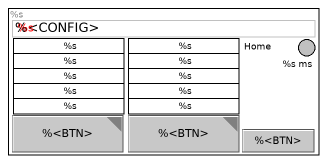
[picture p238: ZLIB_VALVE_5_SENSORS (HMI screen)]
rectangle at (0,0)-(311,147): text "%s"; shows $Object$.BitName
rectangle at (5,30)-(116,46): text "%s"; shows $Object$.SAInitPosName; invisible if $Object$.NoOfInitSensors<1; alarm colour if $Object$.AInitPosition; dynamic style TRUE
rectangle at (5,45)-(116,61): text "%s"; shows $Object$.SBInitPosName; invisible if $Object$.NoOfInitSensors<2; alarm colour if $Object$.BInitPosition; dynamic style TRUE
rectangle at (120,30)-(231,46): text "%s"; shows $Object$.SAWorkPosName; invisible if $Object$.NoOfWorkSensors<1; alarm colour if $Object$.AWorkPosition; dynamic style TRUE
rectangle at (120,45)-(231,61): text "%s"; shows $Object$.SBWorkPosName; invisible if $Object$.NoOfWorkSensors<2; alarm colour if $Object$.BWorkPosition; dynamic style TRUE
ellipse at (290,31)-(307,48): alarm colour if $Object$.HomePosition; dynamic style TRUE
rounded rectangle at (234,32)-(280,45): text "Home"; shows $Object$.State
rectangle at (235,48)-(306,64): text "%s ms"; shows $Object$.ProcessTime
rectangle at (5,60)-(116,76): text "%s"; shows $Object$.SCInitPosName; invisible if $Object$.NoOfInitSensors<3; alarm colour if $Object$.CInitPosition; dynamic style TRUE
rectangle at (120,60)-(231,76): text "%s"; shows $Object$.SCWorkPosName; invisible if $Object$.NoOfWorkSensors<3; alarm colour if $Object$.CWorkPosition; dynamic style TRUE
rectangle at (5,75)-(116,91): text "%s"; shows $Object$.SDInitPosName; invisible if $Object$.NoOfInitSensors<4; alarm colour if $Object$.DInitPosition; dynamic style TRUE
rectangle at (120,75)-(231,91): text "%s"; shows $Object$.SDWorkPosName; invisible if $Object$.NoOfWorkSensors<4; alarm colour if $Object$.DWorkPosition; dynamic style TRUE
rectangle at (5,90)-(116,106): text "%s"; shows $Object$.SEInitPosName; invisible if $Object$.NoOfInitSensors<5; alarm colour if $Object$.EInitPosition; dynamic style TRUE
rectangle at (120,90)-(231,106): text "%s"; shows $Object$.SEWorkPosName; invisible if $Object$.NoOfWorkSensors<5; alarm colour if $Object$.EWorkPosition; dynamic style TRUE
button at (234,121)-(306,144): text "%<BTN>"; shows $Object$.BtnReset.Text; invisible if NOT $Object$.BtnReset.Visible; taps $Object$.BtnReset.Pressed; dynamic style $Object$.BtnReset.TextColor, $Object$.BtnReset.BackgroundColor, $Object$.BtnReset.BackgroundColor, NOT $Object$.BtnReset.Enable
button at (120,107)-(231,144): text "%<BTN>"; shows $Object$.BtnMoveWork.Text; invisible if NOT $Object$.BtnMoveWork.Visible; taps $Object$.BtnMoveWork.Pressed; dynamic style $Object$.BtnMoveWork.TextColor, $Object$.BtnMoveWork.BackgroundColor, $Object$.BtnMoveWork.BackgroundColor, NOT $Object$.BtnMoveWork.Enable
button at (4,107)-(115,144): text "%<BTN>"; shows $Object$.BtnMoveInit.Text; invisible if NOT $Object$.BtnMoveInit.Visible; taps $Object$.BtnMoveInit.Pressed; dynamic style $Object$.BtnMoveInit.TextColor, $Object$.BtnMoveInit.BackgroundColor, $Object$.BtnMoveInit.BackgroundColor, NOT $Object$.BtnMoveInit.Enable
rectangle at (5,11)-(306,28): text "%<CONFIG>"; shows $Object$.InstName
rounded rectangle at (4,12)-(307,29): text "%s"; shows $Object$.ErrorString; invisible if NOT $Object$.ErrorPresent
polygon at (99,109)-(113,123): invisible if $Object$.NoOfValveCoils<2; alarm colour if $Object$.CoilB
polygon at (215,109)-(229,123): alarm colour if $Object$.CoilA
*)

(* Visualisation ZLIB_SERVICELINE
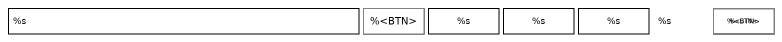
rectangle at (0,0)-(351,26): text "%s"; shows Service.daten[$Object$].Name; editable; dynamic style ST_Service.ColorName[$Object$], $deaktivieren$
embedded screen at (355,0)-(416,26): ZLIB_VISUBUTTON_TOGGELN
rectangle at (495,0)-(566,26): text "%s"; shows Service.daten[$Object$].Warning_Value; editable 0..; dynamic style $deaktivieren$
embedded screen at (705,0)-(766,26): ZLIB_VISUBUTTON
rectangle at (420,0)-(491,26): text "%s"; shows Service.daten[$Object$].Default_Value; editable 0..; dynamic style $deaktivieren$
rectangle at (570,0)-(641,26): text "%s"; shows Service.visu[$Object$].Current_Value; dynamic style Service.visu[$Object$].Current_Value_Color
rectangle at (645,0)-(706,26): text "%s"; shows Service.daten[$Object$].Unit
embedded screen at (705,0)-(766,26): ZLIB_VISUBUTTON_S17
rectangle at (0,0)-(351,26): text "%s"; shows Service.daten[$Object$].Name; invisible if $deaktivieren$; editable; dynamic style ST_Service.ColorName[$Object$], $deaktivieren$
rectangle at (495,0)-(566,26): text "%s"; shows Service.daten[$Object$].Warning_Value; invisible if $deaktivieren$; editable 0..; dynamic style $deaktivieren$
rectangle at (420,0)-(491,26): text "%s"; shows Service.daten[$Object$].Default_Value; invisible if $deaktivieren$; editable 0..; dynamic style $deaktivieren$
*)

(* Visualisation ZLIB_SERVICELIST
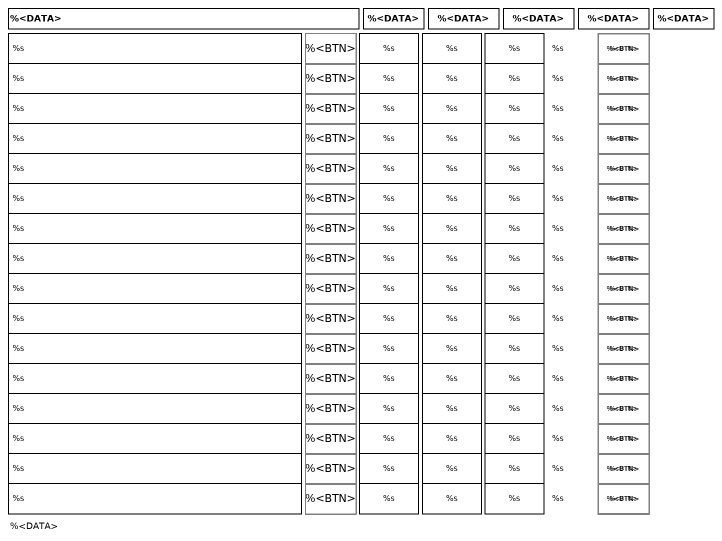
embedded screen at (0,25)-(641,56): ZLIB_SERVICELINE
embedded screen at (0,55)-(641,86): ZLIB_SERVICELINE
rectangle at (0,0)-(351,21): text "%<DATA>"; shows 'Bezeichung der Wartung'
rectangle at (355,0)-(416,21): text "%<DATA>"; shows 'Art'
rectangle at (420,0)-(491,21): text "%<DATA>"; shows 'Vorgabe'
rectangle at (495,0)-(566,21): text "%<DATA>"; shows 'Warngrenze'
rectangle at (570,0)-(641,21): text "%<DATA>"; shows 'Aktuell'
rectangle at (645,0)-(706,21): text "%<DATA>"; shows 'Einheit'
embedded screen at (0,85)-(641,116): ZLIB_SERVICELINE
embedded screen at (0,115)-(641,146): ZLIB_SERVICELINE
embedded screen at (0,145)-(641,176): ZLIB_SERVICELINE
embedded screen at (0,175)-(641,206): ZLIB_SERVICELINE
embedded screen at (0,205)-(641,236): ZLIB_SERVICELINE
embedded screen at (0,235)-(641,266): ZLIB_SERVICELINE
embedded screen at (0,265)-(641,296): ZLIB_SERVICELINE
embedded screen at (0,295)-(641,326): ZLIB_SERVICELINE
embedded screen at (0,325)-(641,356): ZLIB_SERVICELINE
embedded screen at (0,355)-(641,386): ZLIB_SERVICELINE
embedded screen at (0,385)-(641,416): ZLIB_SERVICELINE
embedded screen at (0,415)-(641,446): ZLIB_SERVICELINE
embedded screen at (0,445)-(641,476): ZLIB_SERVICELINE
embedded screen at (0,475)-(641,506): ZLIB_SERVICELINE
rectangle at (0,505)-(766,531): text "%<DATA>"; shows 'Info'
*)

(* Visualisation ZLIB_VISUBUTTON_TOGGELN
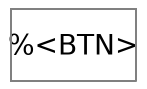
rectangle at (0,0)-(126,73): text "%<BTN>"; shows $Object$.Text; invisible if NOT $Object$.Visible; alarm colour if NOT $Object$.Enable; taps $Object$.Pressed; dynamic style $Object$.TextColor, $Object$.BackgroundColor, $Object$.BackgroundColor, NOT $Object$.Enable
polyline at (125,1)-(125,72): invisible if NOT $Object$.Visible; alarm colour if $Object$.Pressed
polyline at (1,72)-(125,72): invisible if NOT $Object$.Visible; alarm colour if $Object$.Pressed
polyline at (1,1)-(125,1): invisible if NOT $Object$.Visible; alarm colour if NOT $Object$.Pressed
polyline at (1,1)-(1,72): invisible if NOT $Object$.Visible; alarm colour if NOT $Object$.Pressed
polyline at (0,73)-(126,73): invisible if NOT $Object$.Visible; alarm colour if $Object$.Pressed
polyline at (126,0)-(126,73): invisible if NOT $Object$.Visible; alarm colour if $Object$.Pressed
polyline at (0,0)-(126,0): invisible if NOT $Object$.Visible; alarm colour if NOT $Object$.Pressed
polyline at (0,0)-(0,73): invisible if NOT $Object$.Visible; alarm colour if NOT $Object$.Pressed
*)

(* Visualisation INFO_TREE
rounded rectangle at (0,0)-(161,21): text "%<TREE>"; shows $Objekt$.Text; invisible if $Objekt$.unsichtbar; taps $Objekt$.tasten; opens $Objekt$.Zoom; dynamic style $Objekt$.TextFarbe, $Objekt$.deaktivieren
*)

(* Visualisation VISUBUTTON_TREE
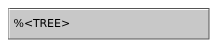
button at (0,0)-(201,31): text "%<TREE>"; shows $Objekt$.Text; invisible if $Objekt$.unsichtbar; taps $Objekt$.tasten; opens $Objekt$.Zoom; dynamic style $Objekt$.TextFarbe, $Objekt$.innenFarbe, $Objekt$.innenFarbe, $Objekt$.deaktivieren
*)

(* Visualisation ZLIB_SFC_STATE
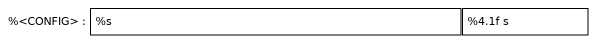
rectangle at (0,0)-(231,27): text "%<CONFIG> :"; shows $SFC$.SFCCurrentPOU
rectangle at (230,0)-(601,27): text "%s"; shows $SFC$.SFCCurrentStep
rectangle at (602,0)-(728,27): text "%4.1f s"; shows $SFC$.SFCTime / 1000.0
*)

(* Visualisation ZLIB_VISUBUTTON
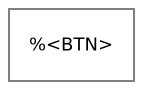
rectangle at (0,0)-(126,73): text "%<BTN>"; shows $Object$.Text; invisible if NOT $Object$.Visible; alarm colour if NOT $Object$.Enable; taps $Object$.Pressed; dynamic style $Object$.TextColor, $Object$.BackgroundColor, $Object$.BackgroundColor, NOT $Object$.Enable
polyline at (125,1)-(125,72): invisible if NOT $Object$.Visible; alarm colour if $Object$.Pressed
polyline at (1,72)-(125,72): invisible if NOT $Object$.Visible; alarm colour if $Object$.Pressed
polyline at (1,1)-(125,1): invisible if NOT $Object$.Visible; alarm colour if NOT $Object$.Pressed
polyline at (1,1)-(1,72): invisible if NOT $Object$.Visible; alarm colour if NOT $Object$.Pressed
polyline at (0,73)-(126,73): invisible if NOT $Object$.Visible; alarm colour if $Object$.Pressed
polyline at (126,0)-(126,73): invisible if NOT $Object$.Visible; alarm colour if $Object$.Pressed
polyline at (0,0)-(126,0): invisible if NOT $Object$.Visible; alarm colour if NOT $Object$.Pressed
polyline at (0,0)-(0,73): invisible if NOT $Object$.Visible; alarm colour if NOT $Object$.Pressed
*)

(* Visualisation ZLIB_VISUBUTTON_ARROW_DOWN
polygon at (2,2)-(102,82): text "%s"; shows $Object$.Text; invisible if NOT $Object$.Visible; alarm colour if NOT $Object$.Enable; taps $Object$.Pressed; dynamic style $Object$.BackgroundColor, $Object$.BackgroundColor, NOT $Object$.Enable
*)

(* Visualisation ZLIB_VISUBUTTON_ARROW_UP
polygon at (2,2)-(102,82): text "%s"; shows $Object$.Text; invisible if NOT $Object$.Visible; alarm colour if NOT $Object$.Enable; taps $Object$.Pressed; dynamic style $Object$.BackgroundColor, $Object$.BackgroundColor, NOT $Object$.Enable
*)

(* Visualisation ZLIB_VISUBUTTON_MODE_SELECT
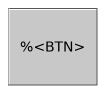
button at (0,0)-(89,77): text "%<BTN>"; shows $Object$.Text; invisible if NOT $Object$.Visible; taps $Object$.Pressed; dynamic style $Object$.TextColor, $Object$.BackgroundColor, $Object$.BackgroundColor, NOT $Object$.Enable
*)

(* Visualisation ZLIB_VISUBUTTON_S17
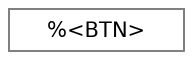
rectangle at (0,0)-(176,43): text "%<BTN>"; shows $Object$.Text; invisible if NOT $Object$.Visible; alarm colour if NOT $Object$.Enable; taps $Object$.Pressed; dynamic style $Object$.TextColor, $Object$.BackgroundColor, $Object$.BackgroundColor, NOT $Object$.Enable
polyline at (175,1)-(175,42): invisible if NOT $Object$.Visible; alarm colour if $Object$.Pressed
polyline at (1,42)-(175,42): invisible if NOT $Object$.Visible; alarm colour if $Object$.Pressed
polyline at (1,1)-(175,1): invisible if NOT $Object$.Visible; alarm colour if NOT $Object$.Pressed
polyline at (1,1)-(1,42): invisible if NOT $Object$.Visible; alarm colour if NOT $Object$.Pressed
polyline at (0,43)-(176,43): invisible if NOT $Object$.Visible; alarm colour if $Object$.Pressed
polyline at (176,0)-(176,43): invisible if NOT $Object$.Visible; alarm colour if $Object$.Pressed
polyline at (0,0)-(176,0): invisible if NOT $Object$.Visible; alarm colour if NOT $Object$.Pressed
polyline at (0,0)-(0,43): invisible if NOT $Object$.Visible; alarm colour if NOT $Object$.Pressed
*)

(* Visualisation ZLIB_VISUBUTTON_S18
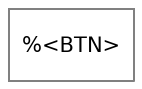
rectangle at (0,0)-(126,73): text "%<BTN>"; shows $Object$.Text; invisible if NOT $Object$.Visible; alarm colour if NOT $Object$.Enable; taps $Object$.Pressed; dynamic style $Object$.TextColor, $Object$.BackgroundColor, $Object$.BackgroundColor, NOT $Object$.Enable
polyline at (125,1)-(125,72): invisible if NOT $Object$.Visible; alarm colour if $Object$.Pressed
polyline at (1,72)-(125,72): invisible if NOT $Object$.Visible; alarm colour if $Object$.Pressed
polyline at (1,1)-(125,1): invisible if NOT $Object$.Visible; alarm colour if NOT $Object$.Pressed
polyline at (1,1)-(1,72): invisible if NOT $Object$.Visible; alarm colour if NOT $Object$.Pressed
polyline at (0,73)-(126,73): invisible if NOT $Object$.Visible; alarm colour if $Object$.Pressed
polyline at (126,0)-(126,73): invisible if NOT $Object$.Visible; alarm colour if $Object$.Pressed
polyline at (0,0)-(126,0): invisible if NOT $Object$.Visible; alarm colour if NOT $Object$.Pressed
polyline at (0,0)-(0,73): invisible if NOT $Object$.Visible; alarm colour if NOT $Object$.Pressed
*)

(* Visualisation ZLIB_VISUBUTTON_S24
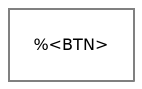
rectangle at (0,0)-(126,73): text "%<BTN>"; shows $Object$.Text; invisible if NOT $Object$.Visible; alarm colour if NOT $Object$.Enable; taps $Object$.Pressed; dynamic style $Object$.TextColor, $Object$.BackgroundColor, $Object$.BackgroundColor, NOT $Object$.Enable
polyline at (125,1)-(125,72): invisible if NOT $Object$.Visible; alarm colour if $Object$.Pressed
polyline at (1,72)-(125,72): invisible if NOT $Object$.Visible; alarm colour if $Object$.Pressed
polyline at (1,1)-(125,1): invisible if NOT $Object$.Visible; alarm colour if NOT $Object$.Pressed
polyline at (1,1)-(1,72): invisible if NOT $Object$.Visible; alarm colour if NOT $Object$.Pressed
polyline at (0,73)-(126,73): invisible if NOT $Object$.Visible; alarm colour if $Object$.Pressed
polyline at (126,0)-(126,73): invisible if NOT $Object$.Visible; alarm colour if $Object$.Pressed
polyline at (0,0)-(126,0): invisible if NOT $Object$.Visible; alarm colour if NOT $Object$.Pressed
polyline at (0,0)-(0,73): invisible if NOT $Object$.Visible; alarm colour if NOT $Object$.Pressed
*)

(* Visualisation ZLIB_VISUBUTTON_S24_S
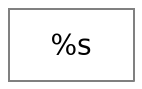
rectangle at (0,0)-(126,73): text "%s"; shows $Object$.Text; invisible if NOT $Object$.Visible; alarm colour if NOT $Object$.Enable; taps $Object$.Pressed; dynamic style $Object$.TextColor, $Object$.BackgroundColor, $Object$.BackgroundColor, NOT $Object$.Enable
polyline at (125,1)-(125,72): invisible if NOT $Object$.Visible; alarm colour if $Object$.Pressed
polyline at (1,72)-(125,72): invisible if NOT $Object$.Visible; alarm colour if $Object$.Pressed
polyline at (1,1)-(125,1): invisible if NOT $Object$.Visible; alarm colour if NOT $Object$.Pressed
polyline at (1,1)-(1,72): invisible if NOT $Object$.Visible; alarm colour if NOT $Object$.Pressed
polyline at (0,73)-(126,73): invisible if NOT $Object$.Visible; alarm colour if $Object$.Pressed
polyline at (126,0)-(126,73): invisible if NOT $Object$.Visible; alarm colour if $Object$.Pressed
polyline at (0,0)-(126,0): invisible if NOT $Object$.Visible; alarm colour if NOT $Object$.Pressed
polyline at (0,0)-(0,73): invisible if NOT $Object$.Visible; alarm colour if NOT $Object$.Pressed
*)

(* Visualisation ZLIB_VISUBUTTON_S24_S_IO
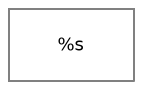
rectangle at (0,0)-(126,73): text "%s"; shows $Object$.Text; invisible if NOT $Object$.Visible; alarm colour if NOT $Object$.Enable; taps $Object$.Pressed; dynamic style $Object$.TextColor, $Object$.BackgroundColor, $Object$.BackgroundColor, NOT $Object$.Enable
polyline at (125,1)-(125,72): invisible if NOT $Object$.Visible; alarm colour if $Object$.Pressed
polyline at (1,72)-(125,72): invisible if NOT $Object$.Visible; alarm colour if $Object$.Pressed
polyline at (1,1)-(125,1): invisible if NOT $Object$.Visible; alarm colour if NOT $Object$.Pressed
polyline at (1,1)-(1,72): invisible if NOT $Object$.Visible; alarm colour if NOT $Object$.Pressed
polyline at (0,73)-(126,73): invisible if NOT $Object$.Visible; alarm colour if $Object$.Pressed
polyline at (126,0)-(126,73): invisible if NOT $Object$.Visible; alarm colour if $Object$.Pressed
polyline at (0,0)-(126,0): invisible if NOT $Object$.Visible; alarm colour if NOT $Object$.Pressed
polyline at (0,0)-(0,73): invisible if NOT $Object$.Visible; alarm colour if NOT $Object$.Pressed
*)

(* Visualisation ZLIB_VISUBUTTON_S36
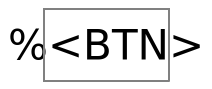
rectangle at (0,0)-(126,73): text "%<BTN>"; shows $Object$.Text; invisible if NOT $Object$.Visible; alarm colour if NOT $Object$.Enable; taps $Object$.Pressed; dynamic style $Object$.TextColor, $Object$.BackgroundColor, $Object$.BackgroundColor, NOT $Object$.Enable
polyline at (125,1)-(125,72): invisible if NOT $Object$.Visible; alarm colour if $Object$.Pressed
polyline at (1,72)-(125,72): invisible if NOT $Object$.Visible; alarm colour if $Object$.Pressed
polyline at (1,1)-(125,1): invisible if NOT $Object$.Visible; alarm colour if NOT $Object$.Pressed
polyline at (1,1)-(1,72): invisible if NOT $Object$.Visible; alarm colour if NOT $Object$.Pressed
polyline at (0,73)-(126,73): invisible if NOT $Object$.Visible; alarm colour if $Object$.Pressed
polyline at (126,0)-(126,73): invisible if NOT $Object$.Visible; alarm colour if $Object$.Pressed
polyline at (0,0)-(126,0): invisible if NOT $Object$.Visible; alarm colour if NOT $Object$.Pressed
polyline at (0,0)-(0,73): invisible if NOT $Object$.Visible; alarm colour if NOT $Object$.Pressed
*)

(* Visualisation ZLIBVISUBUTTON_TEXTINPUT
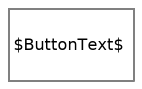
rectangle at (0,0)-(126,73): text "$ButtonText$"; shows $InputVar$; invisible if NOT $Object$.Visible; alarm colour if NOT $Object$.Enable; editable; dynamic style $Object$.TextColor, $Object$.BackgroundColor, $Object$.BackgroundColor, NOT $Object$.Enable
polyline at (125,1)-(125,72): invisible if NOT $Object$.Visible; alarm colour if $Object$.Pressed
polyline at (1,72)-(125,72): invisible if NOT $Object$.Visible; alarm colour if $Object$.Pressed
polyline at (1,1)-(125,1): invisible if NOT $Object$.Visible; alarm colour if NOT $Object$.Pressed
polyline at (1,1)-(1,72): invisible if NOT $Object$.Visible; alarm colour if NOT $Object$.Pressed
polyline at (0,73)-(126,73): invisible if NOT $Object$.Visible; alarm colour if $Object$.Pressed
polyline at (126,0)-(126,73): invisible if NOT $Object$.Visible; alarm colour if $Object$.Pressed
polyline at (0,0)-(126,0): invisible if NOT $Object$.Visible; alarm colour if NOT $Object$.Pressed
polyline at (0,0)-(0,73): invisible if NOT $Object$.Visible; alarm colour if NOT $Object$.Pressed
*)

(* Visualisation ZLIBVISUBUTTON_TEXTVAR
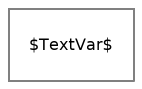
rectangle at (0,0)-(126,73): text "$TextVar$"; shows $TextVar$; invisible if NOT $Object$.Visible; alarm colour if NOT $Object$.Enable; taps $Object$.Pressed; dynamic style $Object$.TextColor, $Object$.BackgroundColor, $Object$.BackgroundColor, NOT $Object$.Enable
polyline at (125,1)-(125,72): invisible if NOT $Object$.Visible; alarm colour if $Object$.Pressed
polyline at (1,72)-(125,72): invisible if NOT $Object$.Visible; alarm colour if $Object$.Pressed
polyline at (1,1)-(125,1): invisible if NOT $Object$.Visible; alarm colour if NOT $Object$.Pressed
polyline at (1,1)-(1,72): invisible if NOT $Object$.Visible; alarm colour if NOT $Object$.Pressed
polyline at (0,73)-(126,73): invisible if NOT $Object$.Visible; alarm colour if $Object$.Pressed
polyline at (126,0)-(126,73): invisible if NOT $Object$.Visible; alarm colour if $Object$.Pressed
polyline at (0,0)-(126,0): invisible if NOT $Object$.Visible; alarm colour if NOT $Object$.Pressed
polyline at (0,0)-(0,73): invisible if NOT $Object$.Visible; alarm colour if NOT $Object$.Pressed
*)

(* Visualisation ZLIBVISUBUTTON_ZOOMTOCALLER
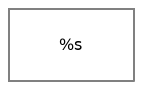
rectangle at (0,0)-(126,73): text "%s"; shows $Object$.Text; invisible if NOT $Object$.Visible; alarm colour if NOT $Object$.Enable; taps $Object$.Pressed; opens ZOOMTOCALLER; dynamic style $Object$.TextColor, $Object$.BackgroundColor, $Object$.BackgroundColor, NOT $Object$.Enable
polyline at (125,1)-(125,72): invisible if NOT $Object$.Visible; alarm colour if $Object$.Pressed
polyline at (1,72)-(125,72): invisible if NOT $Object$.Visible; alarm colour if $Object$.Pressed
polyline at (1,1)-(125,1): invisible if NOT $Object$.Visible; alarm colour if NOT $Object$.Pressed
polyline at (1,1)-(1,72): invisible if NOT $Object$.Visible; alarm colour if NOT $Object$.Pressed
polyline at (0,73)-(126,73): invisible if NOT $Object$.Visible; alarm colour if $Object$.Pressed
polyline at (126,0)-(126,73): invisible if NOT $Object$.Visible; alarm colour if $Object$.Pressed
polyline at (0,0)-(126,0): invisible if NOT $Object$.Visible; alarm colour if NOT $Object$.Pressed
polyline at (0,0)-(0,73): invisible if NOT $Object$.Visible; alarm colour if NOT $Object$.Pressed
*)

(* Visualisation WPC_CONVEYOR_IN
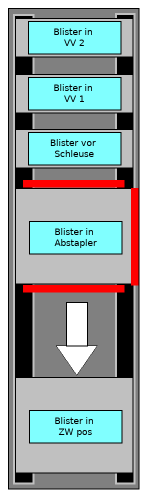
embedded screen at (48,294)-(89,367): SIGNS_ARROWDOWN
rectangle at (7,180)-(125,276): text "%<BASIC>"; shows 'Blister in Abstapler'; alarm colour if NOT ST08_404_B52_2.BitInToCheck; opens Visu.MainMenue.BtnManual_ST08_2.zoom
rectangle at (7,369)-(125,465): text "%<BASIC>"; shows 'Blister in ZW pos'; alarm colour if NOT ST08_406_B54_0.BitInToCheck; opens Visu.MainMenue.BtnManual_ST08_3.zoom
rectangle at (7,121)-(125,160): text "%<BASIC>"; shows 'Blister vor Schleuse'; alarm colour if NOT ST08_402_B51_2.BitInToCheck; opens Visu.MainMenue.BtnManual_ST08_1.zoom
rectangle at (7,66)-(125,105): text "%<BASIC>"; shows 'Blister in VV1'; invisible if NOT .MP.ST08.Trayzufuhr_Verlaengerung; alarm colour if NOT ST08_401_B50_5.BitInToCheck; opens Visu.MainMenue.BtnManual_ST08_1.zoom
rectangle at (7,10)-(125,49): text "%<BASIC>"; shows 'Blister in VV2'; invisible if NOT .MP.ST08.Trayzufuhr_Verlaengerung; alarm colour if NOT ST08_400_B50_0.BitInToCheck; opens Visu.MainMenue.BtnManual_ST08_1.zoom
rectangle at (20,13)-(113,46): text "Blister in / VV 2"; invisible if TRUE
rectangle at (20,69)-(113,102): text "Blister in / VV 1"; invisible if TRUE
rectangle at (20,124)-(113,157): text "Blister vor / Schleuse"; invisible if TRUE
rectangle at (21,213)-(114,246): text "Blister in / Abstapler"; invisible if TRUE
rectangle at (21,402)-(114,435): text "Blister in / ZW pos"; invisible if TRUE
embedded screen at (123,180)-(130,277): DOOR_LOCK; tooltip ST00_229_S1
embedded screen at (15,172)-(116,179): DOOR_LOCK; tooltip ST00_226_S1
embedded screen at (15,277)-(116,284): DOOR_LOCK; tooltip ST00_226_S2
3 more shapes without text or variables
*)

(* Visualisation WPC_CONVEYOR_OUT
embedded screen at (49,4294967295)-(90,72): Signs_ArrowUp
rectangle at (7,61)-(125,100): text "%<BASIC>"; shows 'Stau im Auslauf'; alarm colour if NOT ST08_409_B55_5.BitInToCheck
rectangle at (25,64)-(118,97): text "Stau im / Auslauf"; invisible if TRUE
embedded screen at (7,370)-(129,468): WPC_OUT; shows TD.PartsInBlisterInlet; opens Visu.MainMenue.BtnManual_ST08_3.zoom
embedded screen at (7,183)-(125,284): WPC_OUT_AUFSTAPELN; shows TD.PartsInBlisterInlet; opens Visu.MainMenue.BtnManual_ST08_4.zoom
embedded screen at (7,183)-(14,280): DOOR_LOCK; tooltip ST00_230_S1
embedded screen at (15,176)-(116,183): DOOR_LOCK; tooltip ST00_227_S1
embedded screen at (15,281)-(116,288): DOOR_LOCK; tooltip ST00_227_S2
embedded screen at (0,181)-(7,282): DOOR_LOCK; tooltip ST00_232_S1
3 more shapes without text or variables
*)

(* Visualisation WPC_OUT
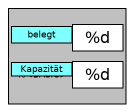
rectangle at (0,0)-(118,96): alarm colour if NOT ST08_406_B54_3.BitInToCheck OR ST08_406_B54_4.ValveSensor
rectangle at (64,16)-(115,43): text "%d"; shows PosIdx-TD.PartsInRoboGripper
rectangle at (2,16)-(64,43): text "%<BASIC>"; shows 'belegt'
rectangle at (64,53)-(115,80): text "%d"; shows TD.PartsInBlisterInlet
rectangle at (2,53)-(64,80): text "%<BASIC>"; shows 'Kapazität'
rectangle at (64,16)-(115,43): shows ST08_CallPRGs.PosIdxHelp; editable 0..TD.PartsInBlisterInlet
rectangle at (3,18)-(64,35): text "belegt"; invisible if TRUE
rectangle at (3,54)-(64,68): text "Kapazität"; invisible if TRUE
rectangle at (64,16)-(115,43): text "%d"; shows PosIdx-TD.PartsInRoboGripper; invisible if $deaktivieren$
*)

(* Visualisation WPC_OUT_AUFSTAPELN
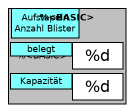
rectangle at (0,0)-(118,96): alarm colour if NOT ST08_407_B55_4.BitInToCheck
rectangle at (2,34)-(64,61): text "%<BASIC>"; shows 'belegt'
rectangle at (64,65)-(115,92): text "%d"; shows .TD.NoOfPalletsPerStack; editable 0..
rectangle at (2,65)-(64,92): text "%<BASIC>"; shows 'Kapazität'
rectangle at (2,34)-(64,48): text "belegt"; invisible if TRUE
rectangle at (2,65)-(64,81): text "Kapazität"; invisible if TRUE
rectangle at (3,0)-(71,30): text "Aufstapeln / Anzahl Blister"; invisible if TRUE
rectangle at (0,3)-(118,31): text "%<BASIC>"; shows 'Aufstapeln Anzahl Blister'
rectangle at (64,34)-(115,61): text "%d"; shows .MP.ST08.NoOfBlisterInStackerOut; editable 0...TD.NoOfPalletsPerStack; dynamic style $deaktivieren$
rectangle at (64,34)-(115,61): text "%d"; shows .MP.ST08.NoOfBlisterInStackerOut; invisible if $deaktivieren$; editable 0...TD.NoOfPalletsPerStack
*)

(* Visualisation ROUNDTABLE
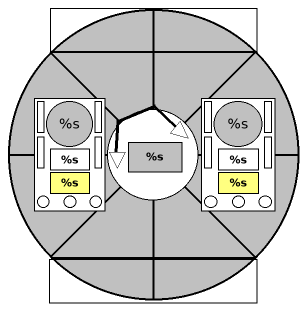
polyline at (147,3)-(147,291): invisible if (ST02_DT_62_B81.ValveSensor OR ST02_DT_62_B91.ValveSensor)
polyline at (2,147)-(292,147): invisible if (ST02_DT_62_B81.ValveSensor OR ST02_DT_62_B91.ValveSensor)
polyline at (44,44)-(249,249): invisible if NOT (ST02_DT_62_B81.ValveSensor OR ST02_DT_62_B91.ValveSensor)
polyline at (44,44)-(249,249): invisible if NOT (ST02_DT_62_B81.ValveSensor OR ST02_DT_62_B91.ValveSensor)
embedded screen at (195,90)-(269,203): RoundTableNest
embedded screen at (28,90)-(99,203): ROUNDTABLENEST
polygon at (103,144)-(119,160): alarm colour if ST02_62_Y6.MoveWork
rounded rectangle at (122,134)-(176,164): text "%s"; shows MachineStates.CycleTimeHelp
polygon at (164,113)-(182,130): alarm colour if ST02_62_Y6.MoveInit
7 more shapes without text or variables
*)

(* Visualisation ROUNDTABLE_1
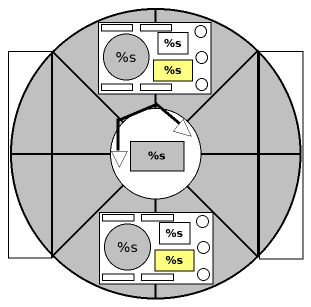
polyline at (147,3)-(147,291): invisible if (ST02_DT_62_B81.ValveSensor OR ST02_DT_62_B91.ValveSensor)
polyline at (2,147)-(292,147): invisible if (ST02_DT_62_B81.ValveSensor OR ST02_DT_62_B91.ValveSensor)
polyline at (44,44)-(249,249): invisible if NOT (ST02_DT_62_B81.ValveSensor OR ST02_DT_62_B91.ValveSensor)
polyline at (44,44)-(249,249): invisible if NOT (ST02_DT_62_B81.ValveSensor OR ST02_DT_62_B91.ValveSensor)
embedded screen at (90,14)-(203,87): RoundTableNest_1
embedded screen at (91,204)-(205,277): ROUNDTABLENEST_1
polygon at (103,144)-(119,160): alarm colour if ST02_62_Y6.MoveWork
rounded rectangle at (122,134)-(176,164): text "%s"; shows MachineStates.CycleTimeHelp
polygon at (165,112)-(183,129): alarm colour if ST02_62_Y6.MoveInit
7 more shapes without text or variables
*)

(* Visualisation ROUNDTABLENEST
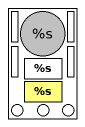
ellipse at (12,3)-(57,48): text "%s"; shows $NestNo$; invisible if NOT MP.ST02.TableData[$NestNo$].ProcessData.Part; alarm colour if MP.ST02.TableData[$NestNo$].ProcessData.Result >11; toggles MP.ST02.TableData[$NestNo$].ProcessData.Part
ellipse at (12,3)-(57,48): text "%s"; shows $NestNo$; invisible if MP.ST02.TableData[$NestNo$].ProcessData.Part; toggles MP.ST02.TableData[$NestNo$].ProcessData.Part
rectangle at (16,73)-(54,94): text "%s"; shows MP.ST02.TableData[$NestNo$].ProcessData.Result; editable
rectangle at (3,38)-(10,69): invisible if NOT MP.ST02.TableData[$NestNo$].ProcessData.Part OR MP.ST02.TableData[$NestNo$].ProcessData.Result >=19; alarm colour if MP.ST02.TableData[$NestNo$].ProcessData.Result >=1
rectangle at (3,3)-(10,34): invisible if NOT MP.ST02.TableData[$NestNo$].ProcessData.Part OR MP.ST02.TableData[$NestNo$].ProcessData.Result >=19; alarm colour if MP.ST02.TableData[$NestNo$].ProcessData.Result >=1
rectangle at (59,38)-(66,69): invisible if NOT MP.ST02.TableData[$NestNo$].ProcessData.Part OR MP.ST02.TableData[$NestNo$].ProcessData.Result >=19; alarm colour if MP.ST02.TableData[$NestNo$].ProcessData.Result >=11
rectangle at (59,3)-(66,34): invisible if NOT MP.ST02.TableData[$NestNo$].ProcessData.Part OR MP.ST02.TableData[$NestNo$].ProcessData.Result >=19; alarm colour if MP.ST02.TableData[$NestNo$].ProcessData.Result >=11
ellipse at (3,96)-(15,108): invisible if MP.ST02.TableData[$NestNo$].ProcessData.Nest_Nr = 0; alarm colour if ST02_Schwenkarm[MP.ST02.TableData[$NestNo$].ProcessData.Nest_Nr].ST02_90_0_sens
ellipse at (29,96)-(41,108): invisible if MP.ST02.TableData[$NestNo$].ProcessData.Nest_Nr = 0; alarm colour if ST02_Schwenkarm[MP.ST02.TableData[$NestNo$].ProcessData.Nest_Nr].ST02_90_sens
ellipse at (54,96)-(66,108): invisible if MP.ST02.TableData[$NestNo$].ProcessData.Nest_Nr = 0; alarm colour if ST02_Schwenkarm[MP.ST02.TableData[$NestNo$].ProcessData.Nest_Nr].ST02_90_180_sens
rectangle at (16,50)-(54,71): text "%s"; shows MP.ST02.TableData[$NestNo$].ProcessData.Nest_Nr; editable 1..2
1 more shapes without text or variables
*)

(* Visualisation ROUNDTABLENEST_1
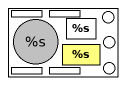
ellipse at (5,12)-(50,57): text "%s"; shows $NestNo$; invisible if NOT MP.ST02.TableData[$NestNo$].ProcessData.Part; alarm colour if MP.ST02.TableData[$NestNo$].ProcessData.Result >=99; toggles MP.ST02.TableData[$NestNo$].ProcessData.Part
ellipse at (5,12)-(50,57): text "%s"; shows $NestNo$; invisible if MP.ST02.TableData[$NestNo$].ProcessData.Part; toggles MP.ST02.TableData[$NestNo$].ProcessData.Part
rectangle at (54,37)-(92,58): text "%s"; shows MP.ST02.TableData[$NestNo$].ProcessData.Result; editable
rectangle at (41,60)-(72,67): invisible if NOT MP.ST02.TableData[$NestNo$].ProcessData.Part OR MP.ST02.TableData[$NestNo$].ProcessData.Result >=19; alarm colour if MP.ST02.TableData[$NestNo$].ProcessData.Result >=1
rectangle at (3,60)-(34,67): invisible if NOT MP.ST02.TableData[$NestNo$].ProcessData.Part OR MP.ST02.TableData[$NestNo$].ProcessData.Result >=19; alarm colour if MP.ST02.TableData[$NestNo$].ProcessData.Result >=1
rectangle at (41,3)-(72,10): invisible if NOT MP.ST02.TableData[$NestNo$].ProcessData.Part OR MP.ST02.TableData[$NestNo$].ProcessData.Result >=19; alarm colour if MP.ST02.TableData[$NestNo$].ProcessData.Result >=11
rectangle at (3,3)-(34,10): invisible if NOT MP.ST02.TableData[$NestNo$].ProcessData.Part OR MP.ST02.TableData[$NestNo$].ProcessData.Result >=19; alarm colour if MP.ST02.TableData[$NestNo$].ProcessData.Result >=11
ellipse at (95,55)-(107,67): invisible if MP.ST02.TableData[$NestNo$].ProcessData.Nest_Nr = 0; alarm colour if ST02_Schwenkarm[MP.ST02.TableData[$NestNo$].ProcessData.Nest_Nr].ST02_90_0_sens
ellipse at (95,29)-(107,41): invisible if MP.ST02.TableData[$NestNo$].ProcessData.Nest_Nr = 0; alarm colour if ST02_Schwenkarm[MP.ST02.TableData[$NestNo$].ProcessData.Nest_Nr].ST02_90_sens
ellipse at (94,4)-(106,16): invisible if MP.ST02.TableData[$NestNo$].ProcessData.Nest_Nr = 0; alarm colour if ST02_Schwenkarm[MP.ST02.TableData[$NestNo$].ProcessData.Nest_Nr].ST02_90_180_sens
rectangle at (58,11)-(88,32): text "%s"; shows MP.ST02.TableData[$NestNo$].ProcessData.Nest_Nr; editable 1..2
1 more shapes without text or variables
*)

(* Visualisation ROUNDTABLENESTNR
ellipse at (0,0)-(45,45): text "%s"; shows MP.ST02.TableData[$NestNo$].ProcessData.Nest_Nr; alarm colour if MP.ST02.DeactivatedNests[MP.ST02.TableData[$NestNo$].ProcessData.Nest_Nr]
*)

(* Visualisation SIGNS_ARROWDOWN
polygon at (0,72)-(48,120): alarm colour if $OnBit$
rectangle at (12,0)-(37,73): alarm colour if $OnBit$
*)

(* Visualisation SIGNS_ARROWLEFT
polygon at (0,0)-(48,48): alarm colour if $OnBit$
rectangle at (48,12)-(121,37): alarm colour if $OnBit$
*)

(* Visualisation SIGNS_ARROWRIGHT
polygon at (72,0)-(120,48): alarm colour if $OnBit$
rectangle at (0,12)-(73,37): alarm colour if $OnBit$
*)

(* Visualisation SIGNS_ARROWUP
polygon at (0,0)-(48,48): alarm colour if $OnBit$
rectangle at (12,48)-(37,121): alarm colour if $OnBit$
*)

(* Visualisation PARTRESULT
